(* PLC project Tc2_MC2_Drive.FB_CoEAX8000DeletePositionOffset Demo, tc3-libraries-kb TwinCAT 3.1 *)
(* stored: creationDateTime 2026-05-21T00:00:00, modificationDateTime 2026-05-21T00:00:00 *)

PROGRAM P_Demo_FB_CoEAX8000DeletePositionOffset
  VAR
    fbAX8000DelOffset : FB_CoEAX8000DeletePositionOffset;  (* AX8000 删位置偏置 FB 实例 *)
    axisServo : AXIS_REF;  (* AX8000 伺服轴轴引用；必须先在 System Manager 配好并 Link *)
    rtDelTrig : R_TRIG;  (* 把电平转上升沿 *)
    bDeleteOffsetReq : BOOL := FALSE;  (* 在线写 TRUE 触发一次删除 *)
    bDelBusy : BOOL;
    bDelError : BOOL;
    nDelErrorID : UDINT;
  END_VAR

// =============================================================================
// 场景：AX8000 驱动的轴维修后要重新做机械找正，先把上一次写进驱动器内存的
//       位置偏置清掉，否则新找正会叠加在旧偏置上导致零点错位。
//
// 价值：1) 偏置常驻 AX8000 侧，要清理时 AX8000 专用 FB 直达
//       2) 也可用硬件无关的 FB_DeletePositionOffset，行为等价
//       3) Memory 选对就只删目标内存里的偏置
//
// !! 注意：Memory 要选偏置实际存放位置，选错会"删了个空"。删偏置改变绝对
//          位置参考，轴静止时删。VAR 含 Position/Relative 字段照常填即可，
//          删除决定权在 Memory。
//
// 验证步骤：
//   1. System Manager 配好 AX8000 NC 轴并 Link 给 axisServo，引用 Tc2_MC2_Drive
//   2. Import PLCopenXML 选本文件，加进 PlcTask，编译登录
//   3. 确认轴静止，确认偏置当初存放在驱动器内存（与本例 Memory 一致）
//   4. 在线写 bDeleteOffsetReq := TRUE → bDelBusy 置 TRUE
//   5. 等 bDelBusy 落回 FALSE 且 bDelError = FALSE 即删除成功
//   6. 若 bDelError = TRUE，看 nDelErrorID 对照 ADS Return Codes 表
// =============================================================================

// 用 R_TRIG 把"持续按住的 TRUE"转成真正的上升沿
rtDelTrig(CLK := bDeleteOffsetReq);

// 单次调用：Memory 选驱动器内存；Axis 是 VAR_IN_OUT 必传
// 本 FB 无 Done，靠 Busy 落回 FALSE 且 Error=FALSE 判成功
fbAX8000DelOffset(
    Execute  := rtDelTrig.Q,
    Position := 0.0,
    Relative := FALSE,
    Feedback := ePositionOffsetFeedback1,
    Memory   := ePositionOffsetMemory_Drive,
    Axis     := axisServo,
    Busy     => bDelBusy,
    Error    => bDelError,
    ErrorID  => nDelErrorID
);
END_PROGRAM
